{attribute 'qualified_only'}
{attribute 'strict'}
TYPE Cover :
(
	FRONT,
	BACK,
	size
);
END_TYPE

(* stored: Version 1.1.0.1, ProductVersion 3.1.4024.11
   DUT Cover: Id {d2ef2d3c-8dc1-4dc9-a0c2-f44fb7befc67} *)
